INTERFACE ITF_Sensor_HMI_Connector EXTENDS ITF_BaseComponent_HMI_Connector

METHOD PUBLIC GetSensorType : E_SensorType
VAR_INPUT
END_VAR
END_METHOD

METHOD PUBLIC GetSensorTypeToString : STRING
END_METHOD

(*			
	EVERDE sp. z o.o.
	Rafał Osajda		05.02.2025		TC 4026.13		wer. 0.0.0.1
	Zwraca aktualny stan czujnika
*)
METHOD IsActive : BOOL
END_METHOD

END_INTERFACE

(* stored: Version 1.1.0.1
   Itf ITF_Sensor_HMI_Connector: Id {57b4f594-d387-4ed4-8db1-68a63d49b635}
   Method GetSensorType: Id {31a21ebe-02ee-4c07-9169-c1701efbd394}
   Method GetSensorTypeToString: Id {590f537c-a25d-49a8-aeac-7b8f8d4b481b}
   Method IsActive: Id {79a44996-4f25-4bd1-b09b-5661b4559709} *)
